Omron CX-Programmer project NuevoProyecto (CX-Programmer 9.61)

# PLC CruceSemaforos: CJ2M CPU31
I/O table (CPU CJ2M-CPU31): rack 0 slot 11 CJ2M-EIP21

## Program NuevoPrograma1 (cyclic task 0)
Local symbols
Amarillo1 1.01 BOOL  ; 1.01
Amarillo2 1.09 BOOL  ; 1.09
Entrada1 0.00 BOOL
Entrada2 0.01 BOOL
P0 2.00 BOOL
P1 2.01 BOOL
P2 2.08 BOOL
P3 2.02 BOOL
P4 2.03 BOOL  ; .
P5 2.04 BOOL
P6 2.05 BOOL
P7 2.06 BOOL
P8 2.07 BOOL
Rojo1 1.00 BOOL  ; 1.00
Rojo2 1.08 BOOL  ; 1.08
Verde1 1.02 BOOL  ; 1.02
Verde2 1.10 BOOL  ; 1.10

### Section Sección1

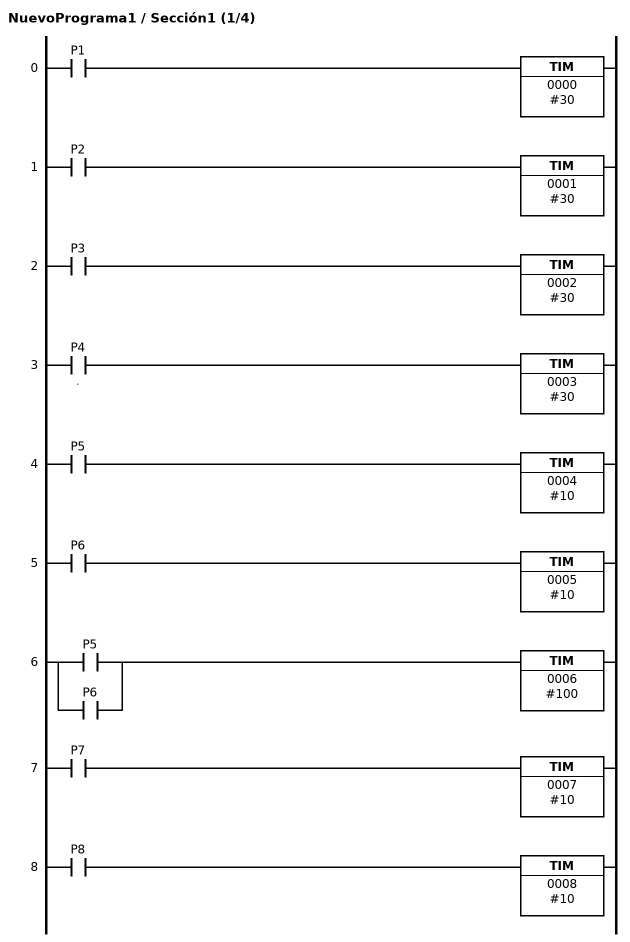
; rung 0
LD P1
TIM 0000 #30
; rung 1
LD P2
TIM 0001 #30
; rung 2
LD P3
TIM 0002 #30
; rung 3
LD P4  ; .
TIM 0003 #30
; rung 4
LD P5
TIM 0004 #10
; rung 5
LD P6
TIM 0005 #10
; rung 6
LD P5
OR P6
TIM 0006 #100
; rung 7
LD P7
TIM 0007 #10
; rung 8
LD P8
TIM 0008 #10

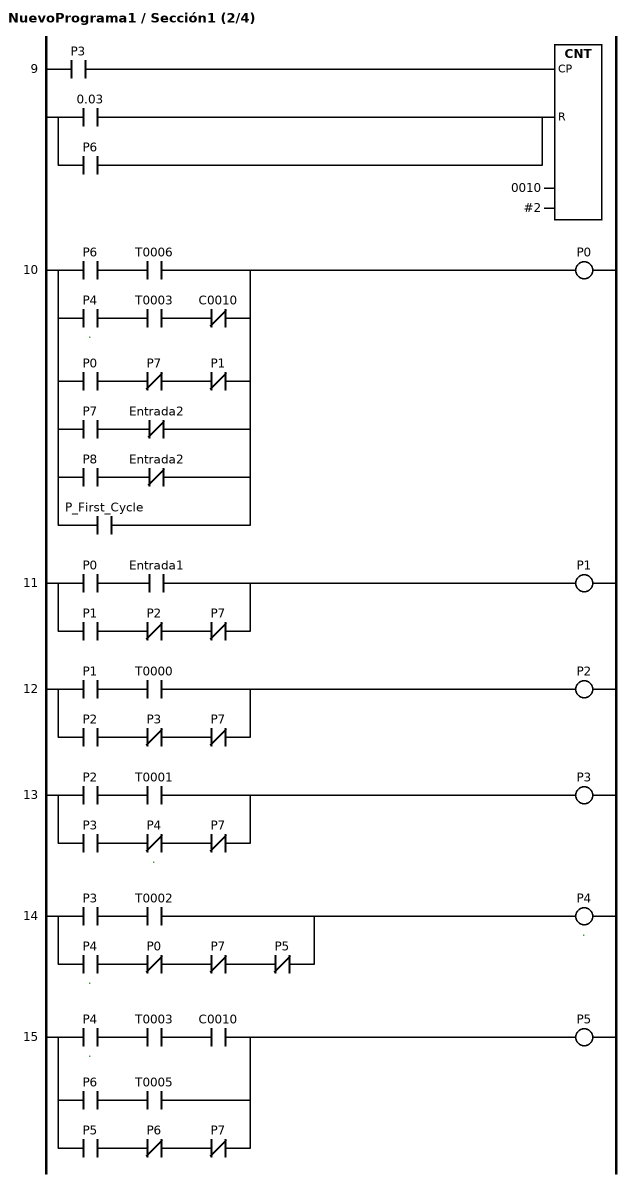
; rung 9
LD P3
LD 0.03
OR P6
CNT 0010 #2
; rung 10
LD P6
AND T0006
LD P4  ; .
AND T0003
ANDNOT C0010
ORLD
LD P0
ANDNOT P7
ANDNOT P1
ORLD
LD P7
ANDNOT Entrada2
ORLD
LD P8
ANDNOT Entrada2
ORLD
OR P_First_Cycle
OUT P0
; rung 11
LD P0
AND Entrada1
LD P1
ANDNOT P2
ANDNOT P7
ORLD
OUT P1
; rung 12
LD P1
AND T0000
LD P2
ANDNOT P3
ANDNOT P7
ORLD
OUT P2
; rung 13
LD P2
AND T0001
LD P3
ANDNOT P4  ; .
ANDNOT P7
ORLD
OUT P3
; rung 14
LD P3
AND T0002
LD P4  ; .
ANDNOT P0
ANDNOT P7
ANDNOT P5
ORLD
OUT P4  ; .
; rung 15
LD P4  ; .
AND T0003
AND C0010
LD P6
AND T0005
ORLD
LD P5
ANDNOT P6
ANDNOT P7
ORLD
OUT P5

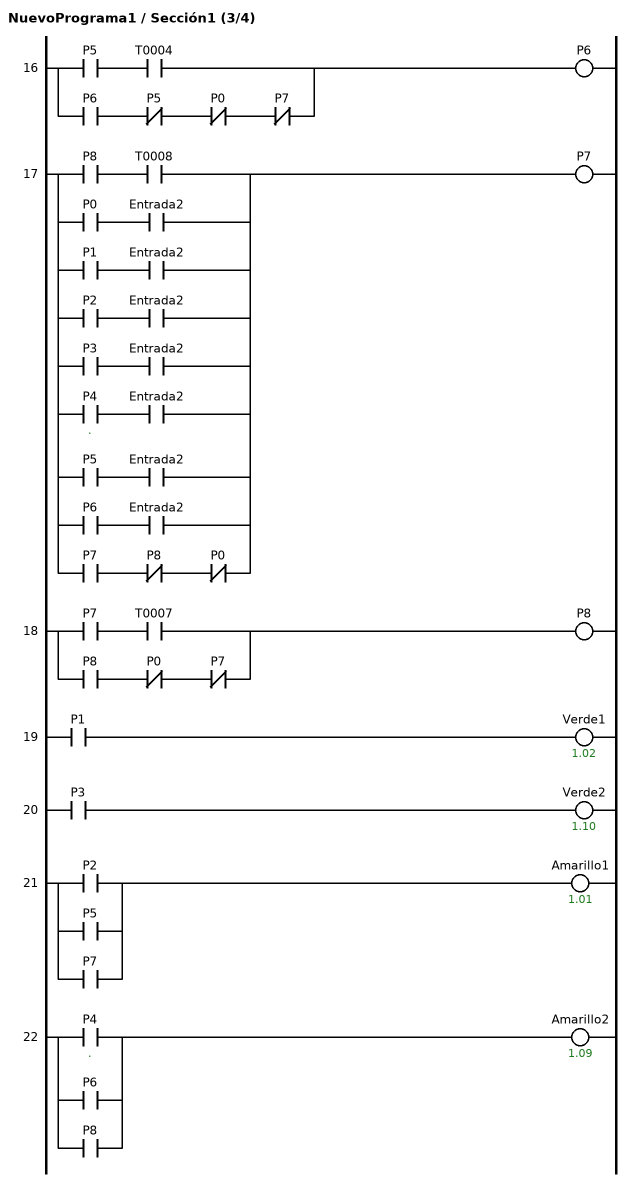
; rung 16
LD P5
AND T0004
LD P6
ANDNOT P5
ANDNOT P0
ANDNOT P7
ORLD
OUT P6
; rung 17
LD P8
AND T0008
LD P0
AND Entrada2
ORLD
LD P1
AND Entrada2
ORLD
LD P2
AND Entrada2
ORLD
LD P3
AND Entrada2
ORLD
LD P4  ; .
AND Entrada2
ORLD
LD P5
AND Entrada2
ORLD
LD P6
AND Entrada2
ORLD
LD P7
ANDNOT P8
ANDNOT P0
ORLD
OUT P7
; rung 18
LD P7
AND T0007
LD P8
ANDNOT P0
ANDNOT P7
ORLD
OUT P8
; rung 19
LD P1
OUT Verde1  ; 1.02
; rung 20
LD P3
OUT Verde2  ; 1.10
; rung 21
LD P2
OR P5
OR P7
OUT Amarillo1  ; 1.01
; rung 22
LD P4  ; .
OR P6
OR P8
OUT Amarillo2  ; 1.09

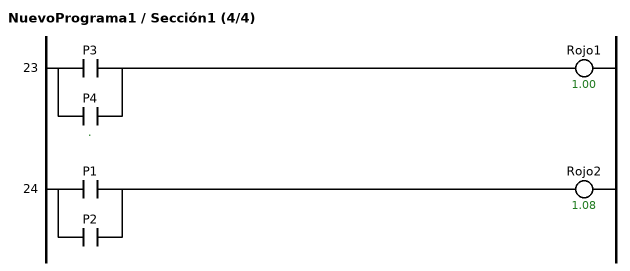
; rung 23
LD P3
OR P4  ; .
OUT Rojo1  ; 1.00
; rung 24
LD P1
OR P2
OUT Rojo2  ; 1.08

### Section END
; rung 0
END(001)